Staubli VAL3: CheckMode.pgx

program CheckMode()
begin
  while !bExit
    nWorkingMode=workingMode(nStatus)
    if nWorkingMode==1
      if nStatus!=0
        resetMotion()
        if taskStatus("Move")==150
          taskResume("Move",1)
          resetMotion()
        endIf
      endIf
    else
      resetMotion()
    endIf
    delay(0)
  endWhile
  resetMotion()
end
